{attribute 'qualified_only'}
{attribute 'strict'}
TYPE E_Buttons :
(
	Start,
	Stop
);
END_TYPE

(* stored: Version 1.1.0.1, ProductVersion 3.1.4024.9
   DUT E_Buttons: Id {94e3f96a-f46b-49a0-a63c-253b3696fcda} *)
